KUKA KRL program: makrosps4.src

&ACCESS RV
&PARAM TEMPLATE = C:\KRC\Roboter\Template\makrospsvorgabe.src
&PARAM EDITMASK = MakroSPS4
&PARAM TPVW_VERSION=8.3.18
DEF MAKROSPS4 ( )
; FOLD Makro Anfang;%{PSE} %MKUKATPVW
SPS_N=-1
; ENDFOLD
; FOLD ;%{H}
END
; ENDFOLD
